(* CoDeSys 2.3.9.31 project: newProject.pr6 *)
(* Libraries: Standard.lib 5.6.98 11:03:02 *)

(* Global variable list: Global_Variables *)
VAR_GLOBAL
	(* Кухня 1 *)
	(* Сенсоры *)
	G_IN_KTN_BTN_1: BOOL; (* Выключатель основной *)
	G_IN_KTN_BTN_2: BOOL; (* Выключатель для вытяжки *)
	G_IN_KTN_DTR_1: BOOL; (* Датчик протечек *)
	(* Реле *)
	G_OUT_KTN_LIGHT_1: BOOL; (* Свет основной *)
	G_OUT_KTN_LIGHT_2: BOOL; (* Свет второстепенный (подсветка) *)
	G_OUT_KTN_FAN_1: BOOL; (* Вытяжка *)

	(* Балкон *)
	(* Сенсоры *)
	G_IN_BLKN_BTN_1: BOOL; (* Выключатель *)
	(* Реле *)
	G_OUT_BLKN_LIGHT_1: BOOL; (* Свет *)

	(* Гостиная *)
	(* Сенсоры *)
	G_IN_LVG_BTN_1: BOOL; (* Выключатель *)
	G_IN_LVG_BTN_2: BOOL; (* Выключатель на рабочем месте *)
	(* Реле *)
	G_OUT_LVG_LIGHT_1: BOOL; (* Свет основной *)
	G_OUT_LVG_LIGHT_2: BOOL; (* Свет второстепенный *)

	(* Спальная *)
	(* Сенсоры *)
	G_IN_BDR_BTN_1: BOOL; (* Выключатель *)
	G_IN_BDR_BTN_2: BOOL; (* Выключатель над кроватью *)
	G_IN_BDR_BTN_3: BOOL; (* Выключатель над кроватью *)
	(* Реле *)
	G_OUT_BDR_LIGHT_1: BOOL; (* Свет *)
	G_OUT_BDR_LIGHT_2: BOOL; (* Свет второстепенный *)
	G_OUT_BDR_LIGHT_3: BOOL; (* Свет над кроватью (торшер) *)
	G_OUT_BDR_LIGHT_4: BOOL; (* Свет над кроватью (торшер) *)

	(* Ванная большая *)
	(* Сенсоры *)
	G_IN_BMB_BTN_1: BOOL; (* Выключатель основной *)
	G_IN_BMB_BTN_2: BOOL; (* Выключатель около зеркала *)
	G_IN_BMB_DTR_1: BOOL; (* Датчик протечек *)
	(* Реле *)
	G_OUT_BMB_LIGHT_1: BOOL; (* Свет основной *)
	G_OUT_BMB_LIGHT_2: BOOL; (* Свет около зеркала *)
	G_OUT_BMB_FAN_1: BOOL; (* Вытяжка *)
	G_OUT_BMB_VLV_1: BOOL; (* Вентиль 1*)
	G_OUT_BMB_VLV_2: BOOL; (* Вентиль 2*)

	(* Детская *)
	(* Сенсоры *)
	G_IN_CHLD_BTN_1: BOOL; (* Выключатель *)
	G_OUT_CHLD_LIGHT_1: BOOL; (* Свет основной *)
	G_OUT_CHLD_LIGHT_2: BOOL; (* Свет второстепенный *)

	(* Коридор *)
	(* Сенсоры *)
	G_IN_HLL_BTN_1: BOOL; (* Проходной выключатель *)
	G_IN_HLL_BTN_2: BOOL; (* Проходной выключатель *)
	G_IN_HLL_BTN_3: BOOL; (* Выключатель на зеркало *)
	G_IN_HLL_DTR_1: BOOL; (* Сенсор открытия двери *)
	G_IN_HLL_DTR_2: BOOL; (* Кнопка звонка *)

	G_OUT_HLL_LIGHT_1: BOOL; (* Свет основной *)
	G_OUT_HLL_LIGHT_2: BOOL; (* Свет второстепенный *)
	G_OUT_HLL_LIGHT_3: BOOL; (* Свет зеркало *)

	(* Ванная малая *)
	(* Сенсоры *)
	G_IN_BMS_BTN_1: BOOL; (* Выключатель *)
	G_IN_BMS_DTR_1: BOOL; (* Датчик протечек *)
	G_OUT_BMS_LIGHT_1: BOOL; (* Вытяжка *)
	G_OUT_BMS_FAN_1: BOOL; (* Вытяжка *)
	G_OUT_BMS_VLV_1: BOOL; (* Вентиль *)
	G_OUT_BMS_VLV_2: BOOL; (* Вентиль *)

	(* Розетки *)
	(* Кухня и балкон *)
	G_OUT_1_2_SOCKET_G1: BOOL; (* Общие *)
	G_OUT_1_2_SOCKET_G2: BOOL; (* Неотключаемые (холодильник)*)
	G_OUT_1_2_SOCKET_G3: BOOL; (* Посудомойка *)
	G_OUT_1_2_SOCKET_G4: BOOL; (* Плита, 380В *)
	(* Гостиная и спальня *)
	G_OUT_3_4_SOCKET_G1: BOOL; (* Общие *)
	G_OUT_3_4_SOCKET_G2: BOOL; (* Неотключаемые (компьютер) *)
	(* Ванная большая *)
	G_OUT_5_SOCKET_G1: BOOL; (* Общие *)
	G_OUT_5_SOCKET_G2: BOOL; (* Стиральная машина *)
	G_OUT_5_SOCKET_G3: BOOL; (* Резерв на бойлер и (или) баню *)
	(* Коридор и детская *)
	G_OUT_6_7_SOCKET_G1: BOOL; (* Общие *)
	G_OUT_6_7_SOCKET_G2: BOOL; (* Неотключаемые (рядом со щитком, роутер, сервер и т.п.) *)

	(* Контроль 0 *)
	G_IN_CTL_BTN_1: BOOL; (* Кнопка ALL *)
	G_IN_CTL_BTN_2: BOOL; (* Кнопка RESET *)
	G_OUT_CTL_ALARM_LAMP: BOOL; (* Лампа-сигнализатор *)
	G_OUT_CTL_ALARM_SOUND: BOOL; (* Зуммер-сигнализатор *)

	(* Переменные для Modbus *)
	ModbusOutVar_0		AT %MW0:	UINT;
	ModbusOutVar_1		AT %MW2:	UINT;
	ModbusOutVar_2		AT %MW4:	UINT;

	ModbusInVar_0		AT %MW6:	UINT;
	ModbusInVar_1		AT %MW8:	UINT;
	ModbusInVar_2		AT %MW10:	UINT;
END_VAR

(* Global variable list: TwinCAT_Import *)
VAR_GLOBAL (* DO NOT CHANGE THIS SHEET MANUALLY! *)

	Term_2_KL2408_1_Output	AT %QX0.0:	BOOL;
	Term_2_KL2408_2_Output	AT %QX0.1:	BOOL;
	Term_2_KL2408_3_Output	AT %QX0.2:	BOOL;
	Term_2_KL2408_4_Output	AT %QX0.3:	BOOL;
	Term_2_KL2408_5_Output	AT %QX0.4:	BOOL;
	Term_2_KL2408_6_Output	AT %QX0.5:	BOOL;
	Term_2_KL2408_7_Output	AT %QX0.6:	BOOL;
	Term_2_KL2408_8_Output	AT %QX0.7:	BOOL;
	Term_3_KL2408_1_Output	AT %QX1.0:	BOOL;
	Term_3_KL2408_2_Output	AT %QX1.1:	BOOL;
	Term_3_KL2408_3_Output	AT %QX1.2:	BOOL;
	Term_3_KL2408_4_Output	AT %QX1.3:	BOOL;
	Term_3_KL2408_5_Output	AT %QX1.4:	BOOL;
	Term_3_KL2408_6_Output	AT %QX1.5:	BOOL;
	Term_3_KL2408_7_Output	AT %QX1.6:	BOOL;
	Term_3_KL2408_8_Output	AT %QX1.7:	BOOL;
	Term_4_KL2408_1_Output	AT %QX2.0:	BOOL;
	Term_4_KL2408_2_Output	AT %QX2.1:	BOOL;
	Term_4_KL2408_3_Output	AT %QX2.2:	BOOL;
	Term_4_KL2408_4_Output	AT %QX2.3:	BOOL;
	Term_4_KL2408_5_Output	AT %QX2.4:	BOOL;
	Term_4_KL2408_6_Output	AT %QX2.5:	BOOL;
	Term_4_KL2408_7_Output	AT %QX2.6:	BOOL;
	Term_4_KL2408_8_Output	AT %QX2.7:	BOOL;
	Term_5_KL2408_1_Output	AT %QX3.0:	BOOL;
	Term_5_KL2408_2_Output	AT %QX3.1:	BOOL;
	Term_5_KL2408_3_Output	AT %QX3.2:	BOOL;
	Term_5_KL2408_4_Output	AT %QX3.3:	BOOL;
	Term_5_KL2408_5_Output	AT %QX3.4:	BOOL;
	Term_5_KL2408_6_Output	AT %QX3.5:	BOOL;
	Term_5_KL2408_7_Output	AT %QX3.6:	BOOL;
	Term_5_KL2408_8_Output	AT %QX3.7:	BOOL;
	Term_6_KL2408_1_Output	AT %QX4.0:	BOOL;
	Term_6_KL2408_2_Output	AT %QX4.1:	BOOL;
	Term_6_KL2408_3_Output	AT %QX4.2:	BOOL;
	Term_6_KL2408_4_Output	AT %QX4.3:	BOOL;
	Term_6_KL2408_5_Output	AT %QX4.4:	BOOL;
	Term_6_KL2408_6_Output	AT %QX4.5:	BOOL;
	Term_6_KL2408_7_Output	AT %QX4.6:	BOOL;
	Term_6_KL2408_8_Output	AT %QX4.7:	BOOL;
	Term_7_KL1408_1_Input	AT %IX0.0:	BOOL;
	Term_7_KL1408_2_Input	AT %IX0.1:	BOOL;
	Term_7_KL1408_3_Input	AT %IX0.2:	BOOL;
	Term_7_KL1408_4_Input	AT %IX0.3:	BOOL;
	Term_7_KL1408_5_Input	AT %IX0.4:	BOOL;
	Term_7_KL1408_6_Input	AT %IX0.5:	BOOL;
	Term_7_KL1408_7_Input	AT %IX0.6:	BOOL;
	Term_7_KL1408_8_Input	AT %IX0.7:	BOOL;
	Term_8_KL1408_1_Input	AT %IX1.0:	BOOL;
	Term_8_KL1408_2_Input	AT %IX1.1:	BOOL;
	Term_8_KL1408_3_Input	AT %IX1.2:	BOOL;
	Term_8_KL1408_4_Input	AT %IX1.3:	BOOL;
	Term_8_KL1408_5_Input	AT %IX1.4:	BOOL;
	Term_8_KL1408_6_Input	AT %IX1.5:	BOOL;
	Term_8_KL1408_7_Input	AT %IX1.6:	BOOL;
	Term_8_KL1408_8_Input	AT %IX1.7:	BOOL;
	Term_9_KL1408_1_Input	AT %IX2.0:	BOOL;
	Term_9_KL1408_2_Input	AT %IX2.1:	BOOL;
	Term_9_KL1408_3_Input	AT %IX2.2:	BOOL;
	Term_9_KL1408_4_Input	AT %IX2.3:	BOOL;
	Term_9_KL1408_5_Input	AT %IX2.4:	BOOL;
	Term_9_KL1408_6_Input	AT %IX2.5:	BOOL;
	Term_9_KL1408_7_Input	AT %IX2.6:	BOOL;
	Term_9_KL1408_8_Input	AT %IX2.7:	BOOL;
	Term_10_KL1408_1_Input	AT %IX3.0:	BOOL;
	Term_10_KL1408_2_Input	AT %IX3.1:	BOOL;
	Term_10_KL1408_3_Input	AT %IX3.2:	BOOL;
	Term_10_KL1408_4_Input	AT %IX3.3:	BOOL;
	Term_10_KL1408_5_Input	AT %IX3.4:	BOOL;
	Term_10_KL1408_6_Input	AT %IX3.5:	BOOL;
	Term_10_KL1408_7_Input	AT %IX3.6:	BOOL;
	Term_10_KL1408_8_Input	AT %IX3.7:	BOOL;
END_VAR

(* POU MAIN, ST *)
PROGRAM MAIN
VAR
	(* Общие переменные *)
	T_LONG_PRESS : TIME := t#1000ms;
	T_LIGHT_OFF : TIME := t#5000ms;
	T_FAN_OFF : TIME := t#10000ms;

	(* Свет и вентиляторы *)
	(* Кухня *)
	KTN_BTN_1 : Z_FB_DIFF_OUT_ON_LONG_AND_SHORT;
	KTN_BTN_2 : Z_FB_SINGLE_SW;
	V_IN_KTN_BTN_MAIN: Z_FB_SINGLE_SW;
	V_IN_KTN_BTN_SUB: Z_FB_SINGLE_SW;
	V_IN_KTN_BTN_FAN: Z_FB_SINGLE_SW;

	(* Балкон *)
	BLKN_BTN : Z_FB_SINGLE_SW;
	V_IN_BLKN_BTN: Z_FB_SINGLE_SW;

	(* Гостиная *)
	LVG_BTN : Z_FB_SHORT_P_OUT1_LONG_P_OUT1_AND_OUT2;
	V_IN_LVG_BTN_MAIN: Z_FB_SINGLE_SW;
	V_IN_LVG_BTN_SUB: Z_FB_SINGLE_SW;

	(* Спальная *)
	BDR_BTN_1 : Z_FB_SHORT_P_OUT1_LONG_P_OUT1_AND_OUT2;
	BDR_BTN_2 : Z_FB_SINGLE_SW;
	BDR_BTN_3 : Z_FB_SINGLE_SW;
	V_IN_BDR_BTN_MAIN: Z_FB_SINGLE_SW;
	V_IN_BDR_BTN_SUB: Z_FB_SINGLE_SW;
	V_IN_BDR_BTN_1: Z_FB_SINGLE_SW;
	V_IN_BDR_BTN_2: Z_FB_SINGLE_SW;

	(* Ванная большая *)
	BMB_BTN_1 : Z_FB_SHRT_P_OUT1_LNG_P_OUT1_OUT2_TIMER;
	BMB_BTN_2 : Z_FB_SINGLE_SW;
	V_IN_BMB_BTN_MAIN: Z_FB_SINGLE_SW;
	V_IN_BMB_BTN_SUB: Z_FB_SINGLE_SW;
	V_IN_BMB_BTN_FAN: Z_FB_SINGLE_SW;

	(* Детская *)
	CHLD_BTN : Z_FB_SHORT_P_OUT1_LONG_P_OUT1_AND_OUT2;
	V_IN_CHLD_BTN_MAIN: Z_FB_SINGLE_SW;
	V_IN_CHLD_BTN_SUB: Z_FB_SINGLE_SW;

	(* Коридор *)
	HLL_BTN_1_2 : FB_HLL; (* Проходные выключатели на основное и подсветку*)
	HLL_BTN_3 : Z_FB_SINGLE_SW_WITH_TIMER; (* Зеркало с таймером *)
	V_IN_HLL_BTN_MAIN: Z_FB_SINGLE_SW;
	V_IN_HLL_BTN_SUB: Z_FB_SINGLE_SW;
	V_IN_HLL_BTN_1: Z_FB_SINGLE_SW;

	(* Ванная малая *)
	BMS_BTN : Z_FB_SHRT_P_OUT1_LNG_P_OUT1_OUT2_TIMER;
	V_IN_BMS_BTN: Z_FB_SINGLE_SW;
	V_IN_BMS_FAN: Z_FB_SINGLE_SW;

	(* Общий выключатель *)
	CTL_BTN_ALL : FB_ALL;

	(* Датчики утечек *)
	IN_WS_LEFT : Z_FB_WS;
	IN_WS_RIGHT : Z_FB_WS;

	(* Обработка тревог  *)
	ALARM : FB_ALARM;
	ERROR : BOOL;

	(* Розетки *)
	(* Кухня и балкон *)
	V_IN_1_2_SOCKET_G1: Z_FB_SINGLE_SW; (* Общие *)
	V_IN_1_2_SOCKET_G2: Z_FB_SINGLE_SW; (* Неотключаемые (холодильник)*)
	V_IN_1_2_SOCKET_G3: Z_FB_SINGLE_SW; (* Посудомойка *)
	V_IN_1_2_SOCKET_G4: Z_FB_SINGLE_SW; (* Плита *)

	(* Гостиная и спальня *)
	V_IN_3_4_SOCKET_G1: Z_FB_SINGLE_SW; (* Общие *)
	V_IN_3_4_SOCKET_G2: Z_FB_SINGLE_SW; (* Неотключаемые (компьютер) *)

	(* Ванная большая *)
	V_IN_5_SOCKET_G1: Z_FB_SINGLE_SW; (* Общие *)
	V_IN_5_SOCKET_G2: Z_FB_SINGLE_SW; (* Стиральная машина *)
	V_IN_5_SOCKET_G3: Z_FB_SINGLE_SW; (* Резерв на бойлер и (или) баню *)

	(* Коридор и детская *)
	V_IN_6_7_SOCKET_G1: Z_FB_SINGLE_SW; (* Общие *)
	V_IN_6_7_SOCKET_G2: Z_FB_SINGLE_SW; (* Неотключаемые (рядом со щитком, роутер, сервер и т.п.) *)

END_VAR
MAP_INPUTS();

(* Кухня *)
(* Кнопка для основного освещения и подсветки *)
KTN_BTN_1 (IN := G_IN_KTN_BTN_1, Q1 := G_OUT_KTN_LIGHT_1, Q2 := G_OUT_KTN_LIGHT_2, TC := T_LONG_PRESS);
(* Кнопка для вентилятора *)
KTN_BTN_2 (IN := G_IN_KTN_BTN_2, Q :=  G_OUT_KTN_FAN_1);
(* Основное освещение  *)
V_IN_KTN_BTN_MAIN(IN := ModbusInVar_0.0, Q := G_OUT_KTN_LIGHT_1);
(* Подсветка *)
V_IN_KTN_BTN_SUB(IN := ModbusInVar_0.1, Q := G_OUT_KTN_LIGHT_2);
 (* Вентилятор *)
V_IN_KTN_BTN_FAN(IN := ModbusInVar_0.2, Q := G_OUT_KTN_FAN_1);

(* Балкон *)
(* Выключатель на балконе *)
BLKN_BTN (IN := G_IN_BLKN_BTN_1, Q := G_OUT_BLKN_LIGHT_1);
V_IN_BLKN_BTN(IN := ModbusInVar_0.3, Q := G_OUT_BLKN_LIGHT_1);

(* Гостиная *)
(* Выключатели проходные *)
LVG_BTN (IN := G_IN_LVG_BTN_1 OR G_IN_LVG_BTN_2, Q1 := G_OUT_LVG_LIGHT_1, Q2 := G_OUT_LVG_LIGHT_2, TC := T_LONG_PRESS);
(* Основное освещение *)
V_IN_LVG_BTN_MAIN(IN := ModbusInVar_0.4, Q := G_OUT_LVG_LIGHT_1);
(* Подсветка *)
V_IN_LVG_BTN_SUB(IN := ModbusInVar_0.5, Q := G_OUT_LVG_LIGHT_2);

(* Спальная *)
(* Выключатели в спальне *)
(* Основной выключатель *)
BDR_BTN_1 (IN := G_IN_BDR_BTN_1, Q1 := G_OUT_BDR_LIGHT_1, Q2 := G_OUT_BDR_LIGHT_2, TC := T_LONG_PRESS);
(* Кнопка у кровати *)
BDR_BTN_2 (IN := G_IN_BDR_BTN_2, Q := G_OUT_BDR_LIGHT_3);
(* Кнопка у кровати *)
BDR_BTN_3 (IN := G_IN_BDR_BTN_3, Q := G_OUT_BDR_LIGHT_4);
(* Основное освещение *)
V_IN_BDR_BTN_MAIN(IN := ModbusInVar_0.6, Q := G_OUT_BDR_LIGHT_1);
(* Подсветка *)
V_IN_BDR_BTN_SUB(IN := ModbusInVar_0.7, Q := G_OUT_BDR_LIGHT_2);
(* Торшер 1 *)
V_IN_BDR_BTN_1(IN := ModbusInVar_0.8, Q := G_OUT_BDR_LIGHT_3);
(* Торшер 2 *)
V_IN_BDR_BTN_2(IN := ModbusInVar_0.9, Q := G_OUT_BDR_LIGHT_4);

(* Ванная большая *)
(* Выключатель основной (освещение и вентилятор)*)
BMB_BTN_1 (IN := G_IN_BMB_BTN_1, Q1 := G_OUT_BMB_LIGHT_1, Q2 := G_OUT_BMB_FAN_1, TC := T_LONG_PRESS, TLight := T_LIGHT_OFF, TFan := T_FAN_OFF);
(* Выключатель зеркало *)
BMB_BTN_2 (IN := G_IN_BMB_BTN_2, Q := G_OUT_BMB_LIGHT_2);
(* Основное освещение *)
V_IN_BMB_BTN_MAIN(IN := ModbusInVar_0.10, Q := G_OUT_BMB_LIGHT_1);
(* Зеркало *)
V_IN_BMB_BTN_SUB(IN := ModbusInVar_0.11, Q := G_OUT_BMB_LIGHT_1);
(* Вентилятор *)
V_IN_BMB_BTN_FAN(IN := ModbusInVar_0.12, Q := G_OUT_BMB_FAN_1);

(* Детская *)
(* Основной выключатель *)
CHLD_BTN (IN := G_IN_CHLD_BTN_1, Q1 := G_OUT_CHLD_LIGHT_1, Q2 := G_OUT_CHLD_LIGHT_2, TC := T_LONG_PRESS);
(* Основное освещение *)
V_IN_CHLD_BTN_MAIN(IN := ModbusInVar_0.13, Q := G_OUT_CHLD_LIGHT_1);
(* Подсветка *)
V_IN_CHLD_BTN_SUB(IN := ModbusInVar_0.14, Q := G_OUT_CHLD_LIGHT_2);

(* Коридор *)
(* Проходные кнопки на основное освещение и подсветку*)
HLL_BTN_1_2 (IN := G_IN_HLL_BTN_1 OR G_IN_HLL_BTN_2, Q1 := G_OUT_HLL_LIGHT_1, Q2 := G_OUT_HLL_LIGHT_2, TC := T_LONG_PRESS);
(* Зеркало *)
HLL_BTN_3 (IN := G_IN_HLL_BTN_3, Q :=G_OUT_HLL_LIGHT_3, TC := T_LIGHT_OFF);
(* Основное освещение *)
V_IN_HLL_BTN_MAIN(IN := ModbusInVar_0.15, Q := G_OUT_HLL_LIGHT_1);
(* Подсветка *)
V_IN_HLL_BTN_SUB(IN := ModbusInVar_1.0, Q := G_OUT_HLL_LIGHT_2);
(* Зеркало *)
V_IN_HLL_BTN_1(IN := ModbusInVar_1.1, Q := G_OUT_HLL_LIGHT_3);

(* Ванная малая *)
(* Выключатель на свет и вентилятор *)
BMS_BTN (IN := G_IN_BMS_BTN_1, M_IN1 := ModbusInVar_1.2, M_IN2 := ModbusInVar_1.3,
	Q1 := G_OUT_BMS_LIGHT_1, Q2 := G_OUT_BMS_FAN_1, TC := T_LONG_PRESS, TLight := T_LIGHT_OFF, TFan := T_FAN_OFF);
(* Основное освещение *)
(*V_IN_BMS_BTN(IN := ModbusInVar_1.2, Q := G_OUT_BMS_LIGHT_1);
(* Вентилятор *)
V_IN_BMS_FAN(IN := ModbusInVar_1.3, Q := G_OUT_BMS_FAN_1);
*)
(* Розетки *)
(* Кухня и балкон *)
(* Общие *)
V_IN_1_2_SOCKET_G1(IN := ModbusInVar_2.0, Q := G_OUT_1_2_SOCKET_G1);
(* Неотключаемые (холодильник)*)
V_IN_1_2_SOCKET_G2(IN := ModbusInVar_2.1, Q := G_OUT_1_2_SOCKET_G2);
(* Посудомойка *)
V_IN_1_2_SOCKET_G3(IN := ModbusInVar_2.2, Q := G_OUT_1_2_SOCKET_G3);
(* Плита *)
V_IN_1_2_SOCKET_G4(IN := ModbusInVar_2.3, Q := G_OUT_1_2_SOCKET_G4);

(* Гостиная и спальня *)
(* Общие *)
V_IN_3_4_SOCKET_G1(IN := ModbusInVar_2.4, Q := G_OUT_3_4_SOCKET_G1);
(* Неотключаемые (компьютер) *)
V_IN_3_4_SOCKET_G2(IN := ModbusInVar_2.5, Q := G_OUT_3_4_SOCKET_G2);

(* Ванная большая *)
(* Общие *)
V_IN_5_SOCKET_G1(IN := ModbusInVar_2.6, Q := G_OUT_5_SOCKET_G1);
(* Стиральная машина *)
V_IN_5_SOCKET_G2(IN := ModbusInVar_2.7, Q := G_OUT_5_SOCKET_G2);
(* Резерв на бойлер и (или) баню *)
V_IN_5_SOCKET_G3(IN := ModbusInVar_2.8, Q := G_OUT_5_SOCKET_G3);

(* Коридор и детская *)
(* Общие *)
V_IN_6_7_SOCKET_G1(IN := ModbusInVar_2.9, Q := G_OUT_6_7_SOCKET_G1);
(* Неотключаемые (рядом со щитком, роутер, сервер и т.п.) *)
V_IN_6_7_SOCKET_G2(IN := ModbusInVar_2.10, Q := G_OUT_6_7_SOCKET_G2);


(* Датчики протечек слева *)
IN_WS_LEFT(IN := G_IN_KTN_DTR_1 OR G_IN_BMS_DTR_1, RESET := G_IN_CTL_BTN_2, Q1 := G_OUT_BMS_VLV_1, Q2 := G_OUT_BMS_VLV_2, ALARM => ERROR);

(* Датчики протечек справа *)
IN_WS_RIGHT(IN := G_IN_BMB_DTR_1, RESET := G_IN_CTL_BTN_2, Q1 := G_OUT_BMB_VLV_1, Q2 := G_OUT_BMB_VLV_2, ALARM => ERROR);

(* Обработка тревоги *)
ALARM(ERROR := ERROR, Q1 := G_OUT_CTL_ALARM_LAMP, Q2 := G_OUT_CTL_ALARM_SOUND);


(* Общий выключатель *)
CTL_BTN_ALL(IN := G_IN_CTL_BTN_1, TC := T_LONG_PRESS);

(* Обработка общего выключателя *)
IF CTL_BTN_ALL.Q1 THEN

	G_OUT_KTN_LIGHT_1 := FALSE;
	G_OUT_KTN_LIGHT_2 := FALSE;
	G_OUT_KTN_FAN_1 := FALSE;

	G_OUT_BLKN_LIGHT_1 := FALSE;

	G_OUT_LVG_LIGHT_1 := FALSE;
	G_OUT_LVG_LIGHT_1 := FALSE;

	G_OUT_BDR_LIGHT_1 := FALSE;
	G_OUT_BDR_LIGHT_2 := FALSE;
	G_OUT_BDR_LIGHT_3 := FALSE;
	G_OUT_BDR_LIGHT_4 := FALSE;

	G_OUT_BMB_LIGHT_1 := FALSE;
	G_OUT_BMB_LIGHT_2 := FALSE;

	G_OUT_CHLD_LIGHT_1 := FALSE;
	G_OUT_CHLD_LIGHT_2 := FALSE;

	G_OUT_HLL_LIGHT_1 := FALSE;
	G_OUT_HLL_LIGHT_2 := FALSE;
	G_OUT_HLL_LIGHT_3 := FALSE;

	G_OUT_BMS_LIGHT_1 := FALSE;
	G_OUT_BMS_FAN_1 := FALSE;

ELSIF CTL_BTN_ALL.Q2 THEN

	G_OUT_1_2_SOCKET_G1 := FALSE;
	G_OUT_1_2_SOCKET_G3 := FALSE;
	G_OUT_1_2_SOCKET_G4 := FALSE;

	G_OUT_3_4_SOCKET_G1 := FALSE;
	G_OUT_3_4_SOCKET_G2 := FALSE;

	G_OUT_5_SOCKET_G1 := FALSE;
	G_OUT_5_SOCKET_G3 := FALSE;

	G_OUT_6_7_SOCKET_G1 := FALSE;

ELSE

	G_OUT_1_2_SOCKET_G1 := CTL_BTN_ALL.G1_STATE;
	(*G_OUT_1_2_SOCKET_G2 := TRUE;
	G_OUT_1_2_SOCKET_G3 := CTL_BTN_ALL.G1_STATE;
	G_OUT_1_2_SOCKET_G4 := CTL_BTN_ALL.G1_STATE;

	G_OUT_3_4_SOCKET_G1 := CTL_BTN_ALL.G1_STATE;
	G_OUT_3_4_SOCKET_G2 := TRUE;

	G_OUT_5_SOCKET_G1 := CTL_BTN_ALL.G1_STATE;
	G_OUT_5_SOCKET_G2 := TRUE;
	G_OUT_5_SOCKET_G3 := CTL_BTN_ALL.G1_STATE;

	G_OUT_6_7_SOCKET_G1 := CTL_BTN_ALL.G1_STATE;
	G_OUT_6_7_SOCKET_G2 := TRUE;*)

END_IF;

MAP_OUTPUTS();
MODBUS_RESET_INPUTS();
MODBUS_SET_OUTPUTS();
END_PROGRAM

(* POU Z_FB_DIFF_OUT_ON_LONG_AND_SHORT, ST *)
(* Обработка длинного и короткого нажатия на два независимых выхода *)
FUNCTION_BLOCK Z_FB_DIFF_OUT_ON_LONG_AND_SHORT
VAR_INPUT
	IN : BOOL;
   	TC : TIME;
END_VAR
VAR_IN_OUT
	Q1 : BOOL;
	Q2 : BOOL;
END_VAR
VAR
	TX : TON;
	MEM1 : BOOL;
	MEM2 : BOOL;
END_VAR
TX(IN := IN, PT := TC);

IF TX.Q AND NOT MEM2 AND IN THEN
	Q2 := NOT Q2;
ELSIF NOT IN AND MEM1 AND NOT MEM2 THEN
	Q1 := NOT Q1;
END_IF;

MEM1 :=  IN;
MEM2 := TX.Q;
END_FUNCTION_BLOCK

(* POU Z_FB_SINGLE_SW, ST *)
(* Кнопка как выключатель *)
FUNCTION_BLOCK Z_FB_SINGLE_SW
VAR_INPUT
	IN: BOOL;
END_VAR
VAR_IN_OUT
	Q: BOOL;
END_VAR
VAR
	MEM : BOOL := FALSE;
END_VAR
IF IN AND NOT MEM THEN
	Q := NOT Q;
END_IF

MEM := IN;
END_FUNCTION_BLOCK

(* POU Z_FB_SHORT_P_OUT1_LONG_P_OUT1_AND_OUT2, ST *)
(* Два выхода
первый - короткое нажатие
первый и второй - длинное нажатие*)
FUNCTION_BLOCK Z_FB_SHORT_P_OUT1_LONG_P_OUT1_AND_OUT2
VAR_INPUT
	IN : BOOL;
   	TC : TIME;
END_VAR
VAR_IN_OUT
	Q1 : BOOL;
	Q2 : BOOL;
END_VAR
VAR
	TX : TON;
	MEM1, MEM2 : BOOL;
END_VAR
TX(IN := IN, PT := TC);

IF IN AND NOT MEM1 THEN
      Q1 := NOT Q1;
      IF NOT Q1 THEN
         Q2 := FALSE;
      END_IF
END_IF

IF TX.Q AND NOT MEM2 AND Q1 THEN
      Q2 := TRUE;
END_IF;

MEM1 := IN;
MEM2 := TX.Q;
END_FUNCTION_BLOCK

(* POU Z_FB_SHRT_P_OUT1_LNG_P_OUT1_OUT2_TIMER, ST *)
(* Два выхода
первый - короткое нажатие
первый и второй - длинное нажатие
при OUT2 = TRUE и длинном нажатии отключается OUT1 и OUT2, 
при OUT1 = TRUE и коротком нажатии отключается OUT1, а OUT2 отключается по таймеру
при OUT1 = TRUE OUT1 отключается по таймеру
*)
FUNCTION_BLOCK Z_FB_SHRT_P_OUT1_LNG_P_OUT1_OUT2_TIMER
VAR_INPUT
	IN : BOOL;
	M_IN1 : BOOL;
	M_IN2 : BOOL;
   	TC : TIME;
	TFan : TIME;
	TLight : TIME;
END_VAR
VAR_IN_OUT
	Q1 : BOOL;
	Q2 : BOOL;
END_VAR
VAR
	TX : TON;
	TPFanInst : TOF;
	TPLightInst : TP;
	MEM1, MEM2 : BOOL;
END_VAR
TX(IN := IN, PT := TC);

IF TX.Q AND NOT MEM2 AND IN THEN
	Q1 := NOT Q1;
	Q2 := NOT Q2;
ELSIF M_IN2 THEN
	Q2 := NOT Q2;
ELSIF (NOT IN AND MEM1 AND NOT MEM2) OR M_IN1 THEN
	Q1 := NOT Q1;
END_IF

TPFanInst(PT := TFan, IN := Q1 OR M_IN2);
IF Q2 AND NOT TPFanInst.Q THEN
	Q2 := TPFanInst.Q;
END_IF

TPLightInst(PT := TLight, IN := Q1 OR M_IN1);
IF Q1 AND NOT TPLightInst.Q THEN
	Q1 := TPLightInst.Q;
	Q2 := TPLightInst.Q;
END_IF

(*AND NOT MEM2 AND IN THEN
	Q2 := NOT Q2;
	Q1 := NOT Q1;
ELSIF NOT IN AND MEM1 THEN
	(*IF NOT MEM2 AND NOT Q2 THEN*)
		Q1 := NOT Q1;
	ELSIF NOT MEM2 AND MEM1 THEN
		Q2 := NOT Q2;
	END_IF;
END_IF;*)

MEM1 :=  IN;
MEM2 := TX.Q;
END_FUNCTION_BLOCK

(* POU FB_HLL, ST *)
FUNCTION_BLOCK FB_HLL
VAR_INPUT
	IN : BOOL;
   	TC : TIME;
END_VAR
VAR_IN_OUT
	Q1 : BOOL;
	Q2 : BOOL;
END_VAR
VAR
	TX : TON;
	MEM1, MEM2 : BOOL;
END_VAR
TX(IN := IN, PT := TC);

IF TX.Q AND NOT MEM2 AND IN THEN
	Q2 := NOT Q2;
ELSIF NOT IN AND MEM1 THEN
	IF NOT MEM2 AND NOT Q2 THEN
		Q1 := NOT Q1;
	ELSIF NOT MEM2 AND MEM1 THEN
		Q2 := NOT Q2;
	END_IF;
END_IF;

MEM1 :=  IN;
MEM2 := TX.Q;
END_FUNCTION_BLOCK

(* POU Z_FB_SINGLE_SW_WITH_TIMER, ST *)
(* Кнопка как выключатель c таймером на отключение *)
FUNCTION_BLOCK Z_FB_SINGLE_SW_WITH_TIMER
VAR_INPUT
	IN: BOOL;
	TC : TIME;
END_VAR
VAR_IN_OUT
	Q: BOOL;
END_VAR
VAR
	MEM : BOOL := FALSE;
	TPInst : TP;
END_VAR
IF IN AND NOT MEM THEN
	Q := NOT Q;
END_IF

TPInst(PT := TC, IN := Q);
IF Q AND NOT TPInst.Q THEN
	Q := TPInst.Q;
END_IF

MEM := IN;
END_FUNCTION_BLOCK

(* POU FB_ALL, ST *)
FUNCTION_BLOCK FB_ALL
VAR_INPUT
	IN: BOOL;
	TC : TIME;
END_VAR
VAR_OUTPUT
	Q1: BOOL := FALSE;
	Q2: BOOL := FALSE;
	G1_STATE: BOOL := TRUE;
END_VAR
VAR
	TX: TON;
	MEM: BOOL;
END_VAR
TX(IN := IN, PT := TC);

IF IN THEN
	IF TX.Q AND NOT MEM THEN
		Q2 := TRUE;
	ELSIF TX.Q AND MEM THEN
		G1_STATE := FALSE;
	ELSIF NOT MEM THEN
		Q1 := TRUE;
		G1_STATE := TRUE;
	END_IF;
ELSE
	Q1 := FALSE;
	Q2 := FALSE;
END_IF;

MEM := TX.Q;
END_FUNCTION_BLOCK

(* POU Z_FB_WS, ST *)
(* Слушаем сенсоры *)
FUNCTION_BLOCK Z_FB_WS
VAR_INPUT
	IN : BOOL;
	RESET : BOOL;
END_VAR
VAR_IN_OUT
	Q1 : BOOL;
	Q2 : BOOL;
END_VAR
VAR_OUTPUT
	ALARM : BOOL := FALSE;
END_VAR
VAR
	MEM : BOOL := FALSE;
END_VAR
IF IN THEN
	Q1 := TRUE;
	Q2 := TRUE;
	ALARM := TRUE;
ELSIF RESET THEN
	Q1 := FALSE;
	Q2 := FALSE;
	ALARM := FALSE;
END_IF

MEM := IN;
END_FUNCTION_BLOCK

(* POU FB_ALARM, ST *)
FUNCTION_BLOCK FB_ALARM
VAR_INPUT
	ERROR : BOOL;
END_VAR
VAR_IN_OUT
	Q1 : BOOL;
	Q2 : BOOL;
END_VAR
VAR
	tProcessTime : TIME;
	tmTimer : TON := (PT:= T#2s);
	Q: BOOL;
END_VAR
IF ERROR THEN
	tmTimer(IN := tProcessTime < T#2S, ET => tProcessTime);
	Q := tProcessTime < T#1S;
ELSE
	Q := FALSE;
END_IF;
Q1 := Q;
Q2 := Q;
END_FUNCTION_BLOCK

(* POU MAP_INPUTS, ST *)
FUNCTION MAP_INPUTS : BOOL
VAR_INPUT
END_VAR
VAR
END_VAR
(* Кухня *)
G_IN_KTN_BTN_1 := Term_7_KL1408_1_Input; (* Выключатель основной *)
G_IN_KTN_BTN_2 := Term_7_KL1408_2_Input; (* Выключатель для вытяжки *)
G_IN_KTN_DTR_1 := Term_9_KL1408_1_Input; (* Датчик протечек *)

(* Балкон *)
G_IN_BLKN_BTN_1 := Term_7_KL1408_3_Input; (* Выключатель *)

(* Гостиная *)
G_IN_LVG_BTN_1 := Term_7_KL1408_4_Input; (* Выключатель *)
G_IN_LVG_BTN_2 := Term_7_KL1408_5_Input; (* Выключатель на рабочем месте *)

(* Спальная *)
G_IN_BDR_BTN_1 := Term_7_KL1408_6_Input; (* Выключатель *)
G_IN_BDR_BTN_2 := Term_7_KL1408_7_Input; (* Выключатель над кроватью *)
G_IN_BDR_BTN_3 := Term_7_KL1408_8_Input; (* Выключатель над кроватью *)

(* Ванная большая *)
G_IN_BMB_BTN_1 := Term_8_KL1408_1_Input; (* Выключатель основной *)
G_IN_BMB_BTN_2 := Term_8_KL1408_2_Input; (* Выключатель около зеркала *)
G_IN_BMB_DTR_1 := Term_9_KL1408_2_Input; (* Датчик протечек *)

(* Детская *)
G_IN_CHLD_BTN_1 := Term_8_KL1408_3_Input; (* Выключатель *)

(* Коридор *)
G_IN_HLL_BTN_1 := Term_8_KL1408_4_Input; (* Проходной выключатель *)
G_IN_HLL_BTN_2 := Term_8_KL1408_5_Input; (* Проходной выключатель *)
G_IN_HLL_BTN_3 := Term_8_KL1408_6_Input; (* Выключатель на зеркало *)
G_IN_HLL_DTR_1 := Term_9_KL1408_3_Input; (* Сенсор открытия двери *)
G_IN_HLL_DTR_2 := Term_9_KL1408_4_Input; (* Кнопка звонка *)

(* Ванная малая *)
G_IN_BMS_BTN_1 := Term_8_KL1408_7_Input; (* Выключатель *)
G_IN_BMS_DTR_1 := Term_9_KL1408_5_Input; (* Датчик протечек *)

(* Контроль *)
G_IN_CTL_BTN_1 := Term_9_KL1408_6_Input; (* Кнопка ALL *)
G_IN_CTL_BTN_2 := Term_9_KL1408_7_Input; (* Кнопка RESET *)
END_FUNCTION

(* POU MAP_OUTPUTS, ST *)
FUNCTION MAP_OUTPUTS : BOOL
VAR_INPUT
END_VAR
VAR
END_VAR
(* Кухня *)
Term_2_KL2408_1_Output := G_OUT_KTN_LIGHT_1; (* Свет основной *)
Term_2_KL2408_2_Output := G_OUT_KTN_LIGHT_2; (* Свет второстепенный (подсветка) *)
Term_2_KL2408_3_Output := G_OUT_KTN_FAN_1; (* Вентилятор *)

(* Балкон *)
Term_2_KL2408_4_Output := G_OUT_BLKN_LIGHT_1; (* Свет *)

(* Гостиная *)
Term_2_KL2408_5_Output := G_OUT_LVG_LIGHT_1; (* Свет основной *)
Term_2_KL2408_6_Output := G_OUT_LVG_LIGHT_2; (* Свет второстепенный *)

(* Спальная *)
Term_2_KL2408_7_Output := G_OUT_BDR_LIGHT_1; (* Свет *)
Term_2_KL2408_8_Output := G_OUT_BDR_LIGHT_2; (* Свет второстепенный *)
Term_3_KL2408_1_Output := G_OUT_BDR_LIGHT_3; (* Свет над кроватью (торшер) *)
Term_3_KL2408_2_Output := G_OUT_BDR_LIGHT_4; (* Свет над кроватью (торшер) *)

(* Ванная большая *)
Term_3_KL2408_3_Output := G_OUT_BMB_LIGHT_1; (* Свет основной *)
Term_3_KL2408_4_Output := G_OUT_BMB_LIGHT_2; (* Свет около зеркала *)
Term_3_KL2408_5_Output := G_OUT_BMB_FAN_1; (* Вытяжка *)
Term_3_KL2408_6_Output := G_OUT_BMB_VLV_1; (* Вентиль *)
Term_3_KL2408_7_Output := G_OUT_BMB_VLV_2; (* Вентиль *)

(* Детская *)
Term_3_KL2408_8_Output := G_OUT_CHLD_LIGHT_1; (* Свет основной *)
Term_4_KL2408_1_Output := G_OUT_CHLD_LIGHT_2; (* Свет второстепенный *)

(* Коридор *)
Term_4_KL2408_2_Output := G_OUT_HLL_LIGHT_1; (* Свет основной *)
Term_4_KL2408_3_Output := G_OUT_HLL_LIGHT_2; (* Свет второстепенный *)
Term_4_KL2408_4_Output := G_OUT_HLL_LIGHT_3; (* Свет зеркало *)

(* Ванная малая *)
Term_4_KL2408_5_Output := G_OUT_BMS_LIGHT_1; (* Свет *)
Term_4_KL2408_6_Output := G_OUT_BMS_FAN_1; (* Вытяжка *)
Term_4_KL2408_7_Output := G_OUT_BMS_VLV_1; (* Вентиль *)
Term_4_KL2408_8_Output := G_OUT_BMS_VLV_2; (* Вентиль *)

(* Контроль *)
Term_5_KL2408_1_Output := G_OUT_CTL_ALARM_LAMP; (* Лампа-сигнализатор *)
Term_5_KL2408_2_Output := G_OUT_CTL_ALARM_SOUND; (* Зуммер-сигнализатор *)

(* Розетки *)
(* Кухня и балкон *)
Term_5_KL2408_3_Output := G_OUT_1_2_SOCKET_G1; (* Общие *)
Term_5_KL2408_4_Output := G_OUT_1_2_SOCKET_G2; (* Неотключаемые (холодильник)*)
Term_5_KL2408_5_Output := G_OUT_1_2_SOCKET_G3; (* Посудомойка *)
Term_5_KL2408_6_Output := G_OUT_1_2_SOCKET_G4; (* Плита, 380В *)
(* Гостиная и спальня *)
Term_5_KL2408_7_Output := G_OUT_3_4_SOCKET_G1; (* Общие *)
Term_5_KL2408_8_Output := G_OUT_3_4_SOCKET_G2; (* Неотключаемые (компьютер) *)
(* Ванная большая *)
Term_6_KL2408_1_Output := G_OUT_5_SOCKET_G1; (* Общие *)
Term_6_KL2408_2_Output := G_OUT_5_SOCKET_G2; (* Стиральная машина *)
Term_6_KL2408_3_Output := G_OUT_5_SOCKET_G3; (* Резерв на бойлер и (или) баню *)
(* Коридор и детская *)
Term_6_KL2408_4_Output := G_OUT_6_7_SOCKET_G1; (* Общие *)
Term_6_KL2408_5_Output := G_OUT_6_7_SOCKET_G2; (* Неотключаемые (рядом со щитком, роутер, сервер и т.п.) *)
END_FUNCTION

(* POU MODBUS_RESET_INPUTS, ST *)
FUNCTION MODBUS_RESET_INPUTS : BOOL
VAR_INPUT
END_VAR
VAR
END_VAR
ModbusInVar_0.0 := FALSE;
ModbusInVar_0.1 := FALSE;
ModbusInVar_0.2 := FALSE;
ModbusInVar_0.3 := FALSE;
ModbusInVar_0.4 := FALSE;
ModbusInVar_0.5 := FALSE;
ModbusInVar_0.6 := FALSE;
ModbusInVar_0.7 := FALSE;
ModbusInVar_0.8 := FALSE;
ModbusInVar_0.9 := FALSE;
ModbusInVar_0.10 := FALSE;
ModbusInVar_0.11 := FALSE;
ModbusInVar_0.12 := FALSE;
ModbusInVar_0.13 := FALSE;
ModbusInVar_0.14 := FALSE;
ModbusInVar_0.15 := FALSE;

ModbusInVar_1.0 := FALSE;
ModbusInVar_1.1 := FALSE;
ModbusInVar_1.2 := FALSE;
ModbusInVar_1.3 := FALSE;
ModbusInVar_1.4 := FALSE;
ModbusInVar_1.5 := FALSE;
ModbusInVar_1.6 := FALSE;
ModbusInVar_1.7 := FALSE;
ModbusInVar_1.8 := FALSE;
ModbusInVar_1.9 := FALSE;
ModbusInVar_1.10 := FALSE;
ModbusInVar_1.11 := FALSE;
ModbusInVar_1.12 := FALSE;
ModbusInVar_1.13 := FALSE;
ModbusInVar_1.14 := FALSE;
ModbusInVar_1.15 := FALSE;

ModbusInVar_2.0 := FALSE;
ModbusInVar_2.1 := FALSE;
ModbusInVar_2.2 := FALSE;
ModbusInVar_2.3 := FALSE;
ModbusInVar_2.4 := FALSE;
ModbusInVar_2.5 := FALSE;
ModbusInVar_2.6 := FALSE;
ModbusInVar_2.7 := FALSE;
ModbusInVar_2.8 := FALSE;
ModbusInVar_2.9 := FALSE;
ModbusInVar_2.10 := FALSE;
ModbusInVar_2.11 := FALSE;
ModbusInVar_2.12 := FALSE;
ModbusInVar_2.13 := FALSE;
ModbusInVar_2.14 := FALSE;
ModbusInVar_2.15 := FALSE;
END_FUNCTION

(* POU MODBUS_SET_OUTPUTS, ST *)
FUNCTION MODBUS_SET_OUTPUTS : BOOL
VAR_INPUT
END_VAR
VAR
END_VAR
ModbusOutVar_0.0 := G_OUT_KTN_LIGHT_1; (*  *)
ModbusOutVar_0.1 := G_OUT_KTN_LIGHT_2; (*  *)
ModbusOutVar_0.2 := G_OUT_KTN_FAN_1; (*  *)
ModbusOutVar_0.3 := G_OUT_BLKN_LIGHT_1; (*  *)
ModbusOutVar_0.4 := G_OUT_LVG_LIGHT_1; (*  *)
ModbusOutVar_0.5 := G_OUT_LVG_LIGHT_2; (*  *)
ModbusOutVar_0.6 := G_OUT_BDR_LIGHT_1; (*  *)
ModbusOutVar_0.7 := G_OUT_BDR_LIGHT_2; (*  *)

ModbusOutVar_0.8 := G_OUT_BDR_LIGHT_3; (*  *)
ModbusOutVar_0.9 := G_OUT_BDR_LIGHT_4; (*  *)
ModbusOutVar_0.10 := G_OUT_BMB_LIGHT_1; (*  *)
ModbusOutVar_0.11 := G_OUT_BMB_LIGHT_2; (*  *)
ModbusOutVar_0.12 := G_OUT_BMB_FAN_1; (*  *)
ModbusOutVar_0.13 := G_OUT_CHLD_LIGHT_1; (*  *)
ModbusOutVar_0.14 := G_OUT_CHLD_LIGHT_2; (*  *)
ModbusOutVar_0.15 := G_OUT_HLL_LIGHT_1; (*  *)

ModbusOutVar_1.0 := G_OUT_HLL_LIGHT_2; (*  *)
ModbusOutVar_1.1 := G_OUT_HLL_LIGHT_3; (*  *)
ModbusOutVar_1.2 := G_OUT_BMS_LIGHT_1; (*  *)
ModbusOutVar_1.3 := G_OUT_BMS_FAN_1; (*  *)
(*
ModbusOutVar_1.4 := ; (*  *)
ModbusOutVar_1.5 := ; (*  *)
ModbusOutVar_1.6 := ; (*  *)
ModbusOutVar_1.7 := ; (*  *)
ModbusOutVar_1.8 := ; (*  *)
*)
ModbusOutVar_1.9 := G_IN_HLL_DTR_1; (*  *)
(*
ModbusOutVar_1.10 := ; (*  *)
ModbusOutVar_1.11 := ; (*  *)
ModbusOutVar_1.12 := ; (*  *)
ModbusOutVar_1.13 := ; (*  *)
ModbusOutVar_1.14 := ; (*  *)
ModbusOutVar_1.15 := ; (*  *)
*)

ModbusOutVar_2.0 := G_OUT_1_2_SOCKET_G1; (*  *)
ModbusOutVar_2.1 := G_OUT_1_2_SOCKET_G2; (*  *)
ModbusOutVar_2.2 := G_OUT_1_2_SOCKET_G3; (*  *)
ModbusOutVar_2.3 := G_OUT_1_2_SOCKET_G4; (*  *)
ModbusOutVar_2.4 := G_OUT_3_4_SOCKET_G1; (*  *)
ModbusOutVar_2.5 := G_OUT_3_4_SOCKET_G2; (*  *)
ModbusOutVar_2.6 := G_OUT_5_SOCKET_G1; (*  *)
ModbusOutVar_2.7 := G_OUT_5_SOCKET_G2; (*  *)
ModbusOutVar_2.8 := G_OUT_5_SOCKET_G3; (*  *)
ModbusOutVar_2.9 := G_OUT_6_7_SOCKET_G1; (*  *)
ModbusOutVar_2.10 := G_OUT_6_7_SOCKET_G2; (*  *)
END_FUNCTION

(* Visualisation TC_VISU
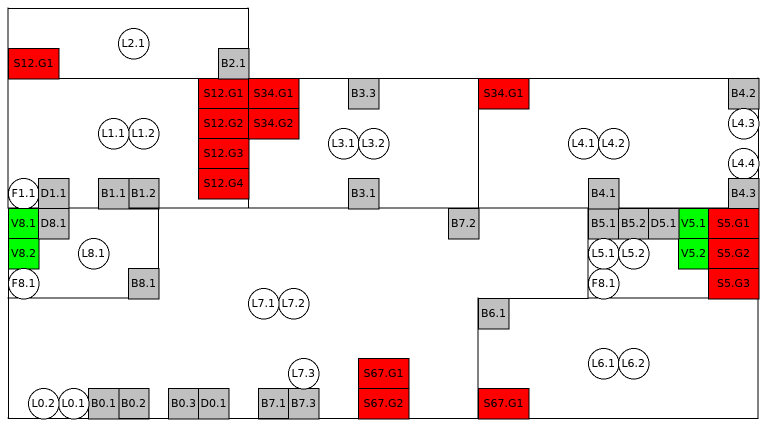
rectangle at (130,180)-(161,211): text "B1.2"; alarm colour if .Term_7_KL1408_2_Input; taps .Term_7_KL1408_2_Input
ellipse at (130,120)-(161,151): text "L1.2"; alarm colour if .G_OUT_KTN_LIGHT_2
ellipse at (100,120)-(131,151): text "L1.1"; alarm colour if .G_OUT_KTN_LIGHT_1
rectangle at (260,390)-(291,421): text "B7.1"; alarm colour if .G_IN_HLL_BTN_1; taps .G_IN_HLL_BTN_1
rectangle at (450,210)-(481,241): text "B7.2"; alarm colour if .G_IN_HLL_BTN_2; taps .G_IN_HLL_BTN_2
rectangle at (120,390)-(151,421): text "B0.2"; alarm colour if .Term_9_KL1408_7_Input; taps .Term_9_KL1408_7_Input
ellipse at (10,180)-(41,211): text "F1.1"; alarm colour if .G_OUT_KTN_FAN_1
rectangle at (200,80)-(251,111): text "S12.G1"; alarm colour if .G_OUT_1_2_SOCKET_G1
rectangle at (200,110)-(251,141): text "S12.G2"; alarm colour if .G_OUT_1_2_SOCKET_G2
rounded rectangle at (40,180)-(71,211): text "D1.1"; alarm colour if .G_IN_KTN_DTR_1; taps .G_IN_KTN_DTR_1
rectangle at (90,390)-(121,421): text "B0.1"; alarm colour if .Term_9_KL1408_6_Input; taps .Term_9_KL1408_6_Input
rectangle at (10,210)-(41,241): text "V8.1"; alarm colour if .G_OUT_BMS_VLV_1
rectangle at (10,240)-(41,271): text "V8.2"; alarm colour if .G_OUT_BMS_VLV_2
rectangle at (350,180)-(381,211): text "B3.1"; alarm colour if .G_IN_LVG_BTN_1; taps .G_IN_LVG_BTN_1
rectangle at (130,270)-(161,301): text "B8.1"; alarm colour if .G_IN_BMS_BTN_1; taps .G_IN_BMS_BTN_1
rectangle at (590,210)-(621,241): text "B5.1"; alarm colour if .G_IN_BMB_BTN_1; taps .G_IN_BMB_BTN_1
rectangle at (680,210)-(711,241): text "V5.1"; alarm colour if .G_OUT_BMB_VLV_1
rectangle at (680,240)-(711,271): text "V5.2"; alarm colour if .G_OUT_BMB_VLV_2
rectangle at (620,210)-(651,241): text "B5.2"; alarm colour if .G_IN_BMB_BTN_2; taps .G_IN_BMB_BTN_2
rounded rectangle at (40,210)-(71,241): text "D8.1"; alarm colour if .G_IN_BMS_DTR_1; taps .G_IN_BMS_DTR_1
rectangle at (100,180)-(131,211): text "B1.1"; alarm colour if .Term_7_KL1408_1_Input; taps .Term_7_KL1408_1_Input
rectangle at (350,80)-(381,111): text "B3.3"; alarm colour if .G_IN_LVG_BTN_2; taps .G_IN_LVG_BTN_2
ellipse at (120,30)-(151,61): text "L2.1"; alarm colour if .G_OUT_BLKN_LIGHT_1
rectangle at (220,50)-(251,81): text "B2.1"; alarm colour if .Term_7_KL1408_3_Input; taps .Term_7_KL1408_3_Input
rectangle at (290,390)-(321,421): text "B7.3"; alarm colour if .G_IN_HLL_BTN_3; taps .G_IN_HLL_BTN_3
rectangle at (170,390)-(201,421): text "B0.3"; alarm colour if .Term_9_KL1408_4_Input; taps .Term_9_KL1408_4_Input
ellipse at (330,130)-(361,161): text "L3.1"; alarm colour if .G_OUT_LVG_LIGHT_1
ellipse at (360,130)-(391,161): text "L3.2"; alarm colour if .G_OUT_LVG_LIGHT_2
rectangle at (590,180)-(621,211): text "B4.1"; alarm colour if .G_IN_BDR_BTN_1; taps .G_IN_BDR_BTN_1
rectangle at (730,80)-(761,111): text "B4.2"; alarm colour if .G_IN_BDR_BTN_2; taps .G_IN_BDR_BTN_2
ellipse at (730,110)-(761,141): text "L4.3"; alarm colour if .G_OUT_BDR_LIGHT_3
ellipse at (730,150)-(761,181): text "L4.4"; alarm colour if .G_OUT_BDR_LIGHT_4
rectangle at (730,180)-(761,211): text "B4.3"; alarm colour if .G_IN_BDR_BTN_3; taps .G_IN_BDR_BTN_3
ellipse at (570,130)-(601,161): text "L4.1"; alarm colour if .G_OUT_BDR_LIGHT_1
ellipse at (600,130)-(631,161): text "L4.2"; alarm colour if .G_OUT_BDR_LIGHT_2
rounded rectangle at (650,210)-(681,241): text "D5.1"; alarm colour if .G_IN_BMB_DTR_1; taps .G_IN_BMB_DTR_1
rectangle at (480,300)-(511,331): text "B6.1"; alarm colour if .G_IN_CHLD_BTN_1; taps .G_IN_CHLD_BTN_1
ellipse at (590,350)-(621,381): text "L6.1"; alarm colour if .G_OUT_CHLD_LIGHT_1
ellipse at (620,350)-(651,381): text "L6.2"; alarm colour if .G_OUT_CHLD_LIGHT_2
ellipse at (280,290)-(311,321): text "L7.2"; alarm colour if .G_OUT_HLL_LIGHT_2
ellipse at (250,290)-(281,321): text "L7.1"; alarm colour if .G_OUT_HLL_LIGHT_1
ellipse at (290,360)-(321,391): text "L7.3"; alarm colour if .G_OUT_HLL_LIGHT_3
ellipse at (60,390)-(91,421): text "L0.1"; alarm colour if .G_OUT_CTL_ALARM_LAMP
rounded rectangle at (200,390)-(231,421): text "D0.1"; alarm colour if .Term_9_KL1408_3_Input; taps .Term_9_KL1408_3_Input
ellipse at (80,240)-(111,271): text "L8.1"; alarm colour if .G_OUT_BMS_LIGHT_1
ellipse at (10,270)-(41,301): text "F8.1"; alarm colour if .G_OUT_BMS_FAN_1
ellipse at (590,270)-(621,301): text "F8.1"; alarm colour if .G_OUT_BMB_FAN_1
ellipse at (30,390)-(61,421): text "L0.2"; alarm colour if .G_OUT_CTL_ALARM_SOUND
ellipse at (590,240)-(621,271): text "L5.1"; alarm colour if .G_OUT_BMB_LIGHT_1
ellipse at (620,240)-(651,271): text "L5.2"; alarm colour if .G_OUT_BMB_LIGHT_2
rectangle at (200,140)-(251,171): text "S12.G3"; alarm colour if .G_OUT_1_2_SOCKET_G3
rectangle at (10,50)-(61,81): text "S12.G1"; alarm colour if .G_OUT_1_2_SOCKET_G1
rectangle at (200,170)-(251,201): text "S12.G4"; alarm colour if .G_OUT_1_2_SOCKET_G4
rectangle at (250,80)-(301,111): text "S34.G1"; alarm colour if .G_OUT_3_4_SOCKET_G1
rectangle at (250,110)-(301,141): text "S34.G2"; alarm colour if .G_OUT_3_4_SOCKET_G2
rectangle at (710,210)-(761,241): text "S5.G1"; alarm colour if .G_OUT_5_SOCKET_G1
rectangle at (710,240)-(761,271): text "S5.G2"; alarm colour if .G_OUT_5_SOCKET_G2
rectangle at (710,270)-(761,301): text "S5.G3"; alarm colour if .G_OUT_5_SOCKET_G3
rectangle at (480,80)-(531,111): text "S34.G1"; alarm colour if .G_OUT_3_4_SOCKET_G1
rectangle at (360,360)-(411,391): text "S67.G1"; alarm colour if .G_OUT_6_7_SOCKET_G1
rectangle at (360,390)-(411,421): text "S67.G2"; alarm colour if .G_OUT_6_7_SOCKET_G2
rectangle at (480,390)-(531,421): text "S67.G1"; alarm colour if .G_OUT_6_7_SOCKET_G1
9 more shapes without text or variables
*)
